PROGRAM F15_AS3_WXT530
VAR
	FB_WXT350_1: FB_WXT350;
	Enable:BOOL:=TRUE;
	FB_FL0: FB_FL;
	ComError :BOOL;
	
	TOF_0: TOF;
END_VAR


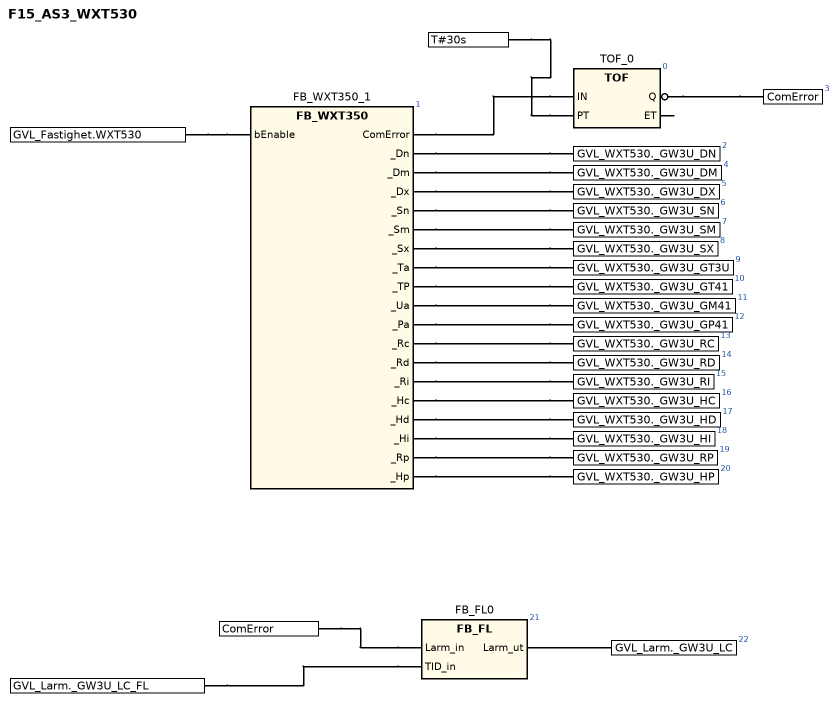
// PAGE
TOF_0(IN := FB_WXT350_1.ComError, PT := T#30s); // TOF
FB_WXT350_1(bEnable := GVL_Fastighet.WXT530); // FB_WXT350
GVL_WXT530._GW3U_DN := FB_WXT350_1._Dn;
ComError := NOT TOF_0.Q;
GVL_WXT530._GW3U_DM := FB_WXT350_1._Dm;
GVL_WXT530._GW3U_DX := FB_WXT350_1._Dx;
GVL_WXT530._GW3U_SN := FB_WXT350_1._Sn;
GVL_WXT530._GW3U_SM := FB_WXT350_1._Sm;
GVL_WXT530._GW3U_SX := FB_WXT350_1._Sx;
GVL_WXT530._GW3U_GT3U := FB_WXT350_1._Ta;
GVL_WXT530._GW3U_GT41 := FB_WXT350_1._TP;
GVL_WXT530._GW3U_GM41 := FB_WXT350_1._Ua;
GVL_WXT530._GW3U_GP41 := FB_WXT350_1._Pa;
GVL_WXT530._GW3U_RC := FB_WXT350_1._Rc;
GVL_WXT530._GW3U_RD := FB_WXT350_1._Rd;
GVL_WXT530._GW3U_RI := FB_WXT350_1._Ri;
GVL_WXT530._GW3U_HC := FB_WXT350_1._Hc;
GVL_WXT530._GW3U_HD := FB_WXT350_1._Hd;
GVL_WXT530._GW3U_HI := FB_WXT350_1._Hi;
GVL_WXT530._GW3U_RP := FB_WXT350_1._Rp;
GVL_WXT530._GW3U_HP := FB_WXT350_1._Hp;
FB_FL0(Larm_in := ComError, TID_in := GVL_Larm._GW3U_LC_FL); // FB_FL
GVL_Larm._GW3U_LC := FB_FL0.Larm_ut;

END_PROGRAM

(* stored: Version 1.1.0.1, ProductVersion 3.1.4022.3
   POU F15_AS3_WXT530: Id {26e9fa4a-c2a0-4127-950d-cc918fa40864}, SpecialFunc None *)
